{attribute 'qualified_only'}
VAR_GLOBAL
	//To Unreal engine
	FpistonMainBoom : LREAL;
	FpistonKnuckleJib : LREAL;
	FpistonKingRotation : LREAL;
	
	
	//From Unreal engine
	VpistonMainBoom : LREAL;
	VpistonKnuckleJib : LREAL;
	VpistonKingRotation : LREAL;
	
	XpistonMainBoom : LREAL;
	XpistonKnuckleJib : LREAL;
	XpistonKingRotation : LREAL;
END_VAR

(* stored: Version 1.1.0.1, ProductVersion 3.1.4024.9
   GVL Work: Id {5ed653ee-4ae3-47db-9070-5b8ede254b65} *)
